// SIMATIC S7-200 project (STEP 7-Micro/WIN), CPU 212 REL 01.00

SYMBOL_TABLE USER1
S1               I0.0     // PULSANTE START
S2               I0.1     // PULSANTE STOP
SPP1             I0.2     // SENSORE SPP1
SPP2             I0.3     // SESNORE SPP2
SPP3             I0.4     // SENSORE SPP3
SGIU             I0.5     // SENSORE TIMBRO GIU
SSU              I0.6     // SENSORE TIMBRO SU
S3               I0.7     // PULSANTE RESET
L                Q0.0     // LAMPADA SEGNALATORE
M                Q0.1     // KM1 CONTATORE MOTORE
EVGIU            Q0.2     // ELETTROVALVOLA GIU
EVSU             Q0.3     // ELETTROVALVOLA SU
END_SYMBOL_TABLE

ORGANIZATION_BLOCK MAIN:OB1
TITLE=PROGRAM COMMENTS
BEGIN
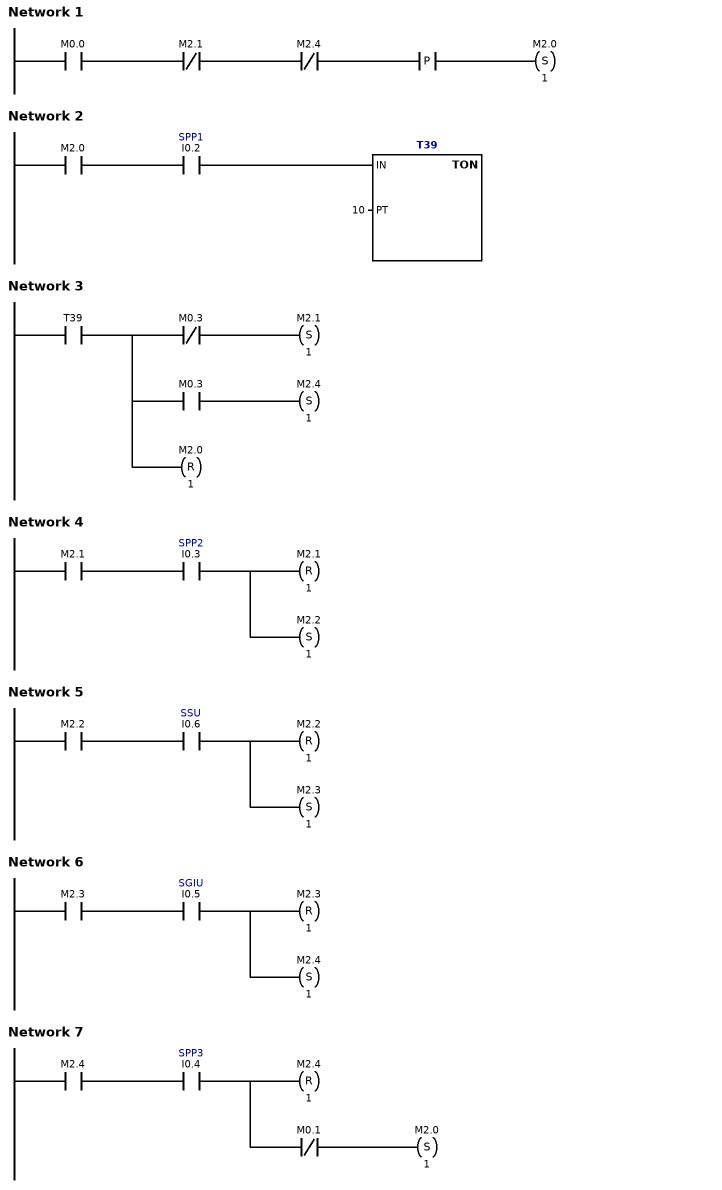
Network 1
LD     M0.0
AN     M2.1
AN     M2.4
EU
S      M2.0, 1
Network 2
LD     M2.0
A      SPP1:I0.2
TON    T39, 10
Network 3
LD     T39
LPS
AN     M0.3
S      M2.1, 1
LRD
A      M0.3
S      M2.4, 1
LPP
R      M2.0, 1
Network 4
LD     M2.1
A      SPP2:I0.3
R      M2.1, 1
S      M2.2, 1
Network 5
LD     M2.2
A      SSU:I0.6
R      M2.2, 1
S      M2.3, 1
Network 6
LD     M2.3
A      SGIU:I0.5
R      M2.3, 1
S      M2.4, 1
Network 7
LD     M2.4
A      SPP3:I0.4
R      M2.4, 1
AN     M0.1
S      M2.0, 1
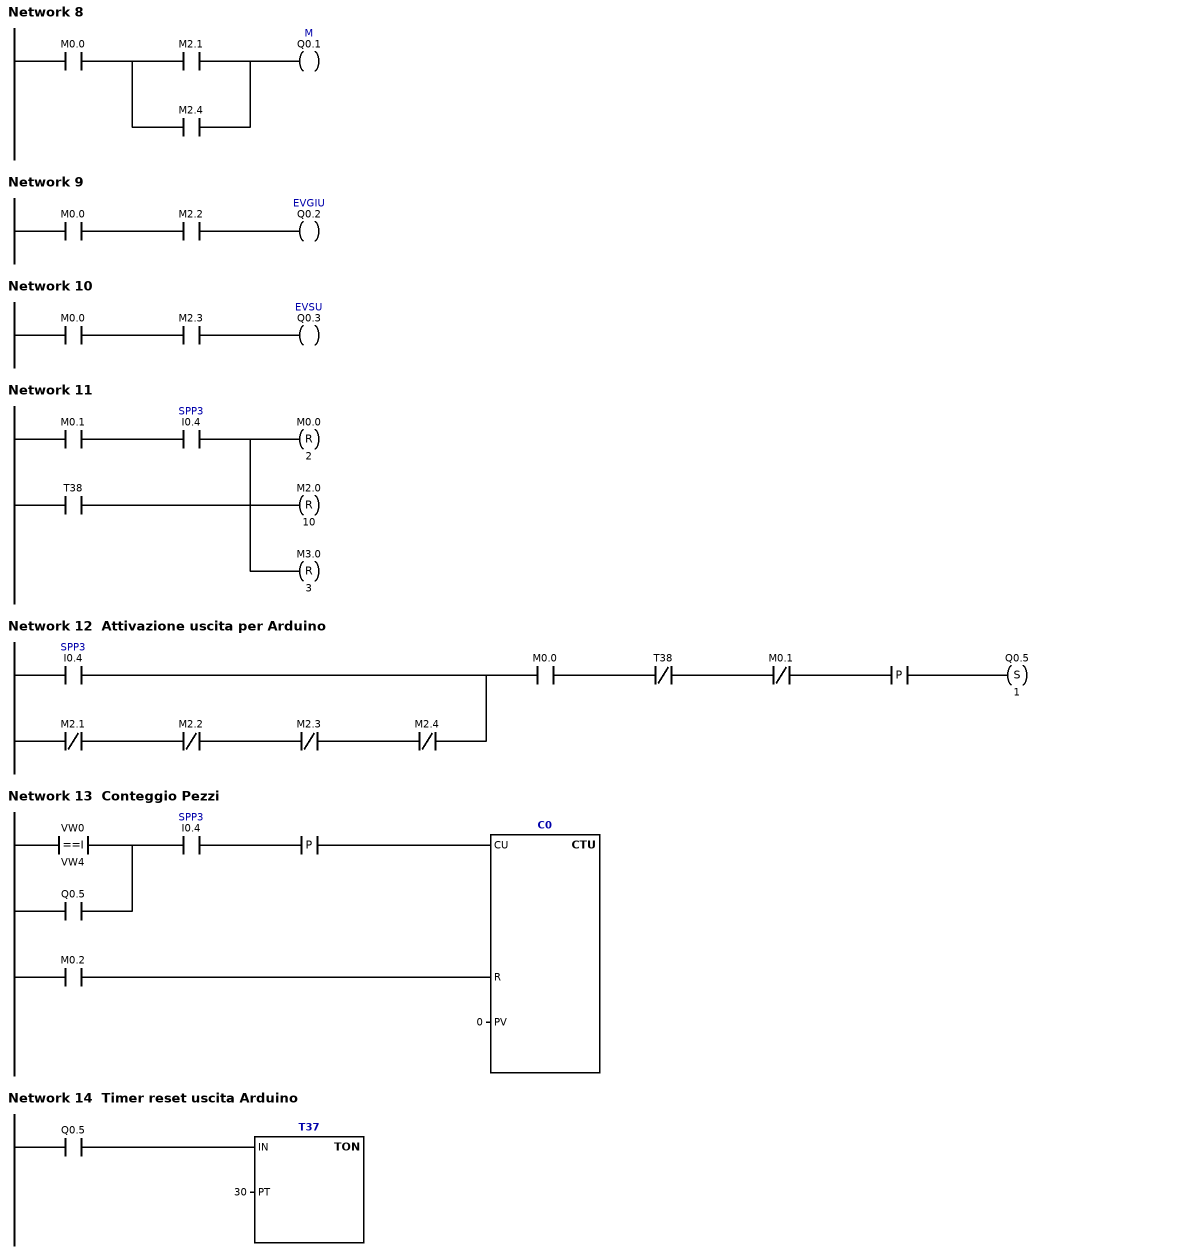
Network 8
LD     M0.0
LD     M2.1
O      M2.4
ALD
=      M:Q0.1
Network 9
LD     M0.0
A      M2.2
=      EVGIU:Q0.2
Network 10
LD     M0.0
A      M2.3
=      EVSU:Q0.3
Network 11
LD     M0.1
A      SPP3:I0.4
O      T38
R      M0.0, 2
R      M2.0, 10
R      M3.0, 3
Network 12 // Attivazione uscita per Arduino
LD     SPP3:I0.4
LDN    M2.1
AN     M2.2
AN     M2.3
AN     M2.4
OLD
A      M0.0
AN     T38
AN     M0.1
EU
S      Q0.5, 1
Network 13 // Conteggio Pezzi
LDW=   VW0, VW4
O      Q0.5
A      SPP3:I0.4
EU
LD     M0.2
CTU    C0, 0
Network 14 // Timer reset uscita Arduino
LD     Q0.5
TON    T37, 30
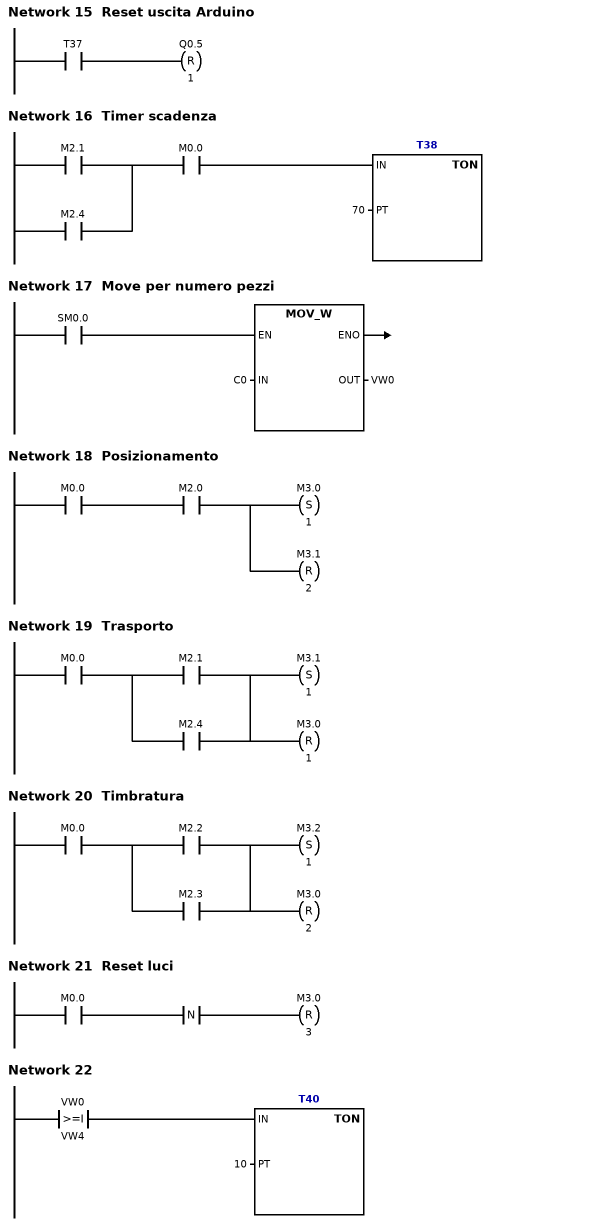
Network 15 // Reset uscita Arduino
LD     T37
R      Q0.5, 1
Network 16 // Timer scadenza
LD     M2.1
O      M2.4
A      M0.0
TON    T38, 70
Network 17 // Move per numero pezzi
LD     SM0.0
MOVW   C0, VW0
Network 18 // Posizionamento
LD     M0.0
A      M2.0
S      M3.0, 1
R      M3.1, 2
Network 19 // Trasporto
LD     M0.0
LD     M2.1
O      M2.4
ALD
S      M3.1, 1
R      M3.0, 1
Network 20 // Timbratura
LD     M0.0
LD     M2.2
O      M2.3
ALD
S      M3.2, 1
R      M3.0, 2
Network 21 // Reset luci
LD     M0.0
ED
R      M3.0, 3
Network 22
LDW>=  VW0, VW4
TON    T40, 10
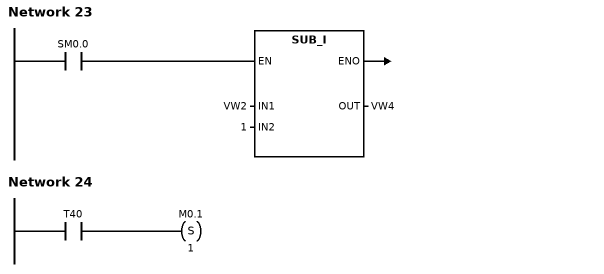
Network 23
LD     SM0.0
MOVW   VW2, VW4
-I     1, VW4
Network 24
LD     T40
S      M0.1, 1
END_ORGANIZATION_BLOCK
